# EPICS substitutions: epics/m-epics-eemcu/eemcuApp/Db/Sim8-m5.substitutions
file "eemcu.template" {
pattern {P,       N,  M,   R,      DTYP,         PORT,     ADDR,  DESC,          EGU, DIR,  VELO, HVEL, JVEL,  JAR,  VBAS,  ACCL,  BDST, DLY,  BVEL,  BACC,  MRES,      ERES,       PREC,  DLLM,  DHLM,  INIT}
{"IOC:",   5,  m5,  m5-,    "asynMotor",   MCU1,     5,     "motor 5",    mm,  Pos,  24.9, 5.05, 10,    10.2, 0,     1,     0,    0.3,  1,     .2,    0.0046875  0.01754386  3,     -140,   13,    ""}
}
